{attribute 'GeneratedUsingTerminal: EL3783-0000-0018'}
{attribute addProperty BoxType "EL3783-0000-0018"}
{attribute addProperty Id "I3_SamplesAT %I*I3_Samples_1109DCAA40"}
{attribute addProperty CRC "1355657212"}
{attribute addProperty Size "40"}
TYPE L3_Current_Samples_50CDAFFC :
STRUCT
	{attribute addProperty Name "I3_Samples"}
	I3_Samples AT %I* : I3_Samples_1109DCAA;
END_STRUCT
END_TYPE

(* stored: Version 1.2.0.0, ProductVersion 3.1.4024.9
   DUT L3_Current_Samples_50CDAFFC: Id {2bfe113c-45ba-4cd2-876e-f531f84063f2} *)
